Staubli VAL3: add.pgx

public program add(num& x_nMatrix1[] (dimensions=2), num& x_nMatrix2[] (dimensions=2), num& x_nResult[] (dimensions=2))
  local num l_nX
  local num l_nY
begin

  resize(x_nResult,1,size(x_nMatrix1,1))
  resize(x_nResult,2,size(x_nMatrix1,2))

  for l_nX = 0 to size(x_nMatrix1,1)-1
    for l_nY = 0 to size(x_nMatrix1,2)-1
      x_nResult[l_nX,l_nY] = x_nMatrix1[l_nX,l_nY] + x_nMatrix2[l_nX,l_nY]
    endFor
  endFor


end
